(* PLC project Untitled1, Beckhoff Automation GmbH TF6420 Database Server Query Analyser 1.0.0.0 *)
(* stored: creationDateTime 2021-11-04T11:13:41, modificationDateTime 2021-11-04T11:13:41 *)

TYPE ST_Record : STRUCT
  ID : LINT;
  Timestamp : DT;
  Name : STRING(80);
  nSensor1 : LREAL;
  nSensor2 : LREAL;
END_STRUCT;
END_TYPE
